# EPICS substitutions: viocs/si_ps/si_psApp/Db/qf3.substitutions
file "db/individual.db" {
    pattern { family, pos }
        { "QF3", "01C2" }
        { "QF3", "01C4" }
        { "QF3", "02C2" }
        { "QF3", "02C4" }
        { "QF3", "03C2" }
        { "QF3", "03C4" }
        { "QF3", "04C2" }
        { "QF3", "04C4" }
        { "QF3", "05C2" }
        { "QF3", "05C4" }
        { "QF3", "06C2" }
        { "QF3", "06C4" }
        { "QF3", "07C2" }
        { "QF3", "07C4" }
        { "QF3", "08C2" }
        { "QF3", "08C4" }
        { "QF3", "09C2" }
        { "QF3", "09C4" }
        { "QF3", "10C2" }
        { "QF3", "10C4" }
        { "QF3", "11C2" }
        { "QF3", "11C4" }
        { "QF3", "12C2" }
        { "QF3", "12C4" }
        { "QF3", "13C2" }
        { "QF3", "13C4" }
        { "QF3", "14C2" }
        { "QF3", "14C4" }
        { "QF3", "15C2" }
        { "QF3", "15C4" }
        { "QF3", "16C2" }
        { "QF3", "16C4" }
        { "QF3", "17C2" }
        { "QF3", "17C4" }
        { "QF3", "18C2" }
        { "QF3", "18C4" }
        { "QF3", "19C2" }
        { "QF3", "19C4" }
        { "QF3", "20C2" }
        { "QF3", "20C4" }
}
